{attribute 'qualified_only'}
VAR_GLOBAL
	OutputData AT %Q*: ARRAY[0..7] OF BYTE;
	
	InputData1 AT %I*: ARRAY[0..7] OF BYTE;
	InputData2 AT %I*: ARRAY[0..7] OF BYTE;
	InputData3 AT %I*: ARRAY[0..7] OF BYTE;
	state AT %I* : UINT;
	
	EHWTable1XML : STRING[6000];

	TrackSegmentsRaw1 : ARRAY[0..29] OF ST_Track_Segment_Raw_EHC:= [
		(iTrackNumber := 1, iXPosition := 0, sType := "straight", sBatch := "B", iId := 61, iLength := 4, rStartValue := 640.0, rEndValue := 644.0),
(iTrackNumber := 2, iXPosition := 4, sType := "straight", sBatch := "B", iId := 58, iLength := 4, rStartValue := 628.0, rEndValue := 632.0),
(iTrackNumber := 3, iXPosition := 8, sType := "straight", sBatch := "B", iId := 60, iLength := 4, rStartValue := 636.0, rEndValue := 640.0),
(iTrackNumber := 4, iXPosition := 12, sType := "straight", sBatch := "B", iId := 24, iLength := 4.2, rStartValue := 304.6, rEndValue := 308.8),
(iTrackNumber := 5, iXPosition := 16.4, sType := "straight", sBatch := "B", iId := 2, iLength := 4.2, rStartValue := 212.2, rEndValue := 216.4),
(iTrackNumber := 6, iXPosition := 20.6, sType := "straight", sBatch := "B", iId := 66, iLength := 4, rStartValue := 660.0, rEndValue := 664.0),
(iTrackNumber := 7, iXPosition := 24.6, sType := "straight", sBatch := "B", iId := 65, iLength := 4, rStartValue := 656.0, rEndValue := 660.0),
(iTrackNumber := 8, iXPosition := 28.6, sType := "straight", sBatch := "B", iId := 55, iLength := 4, rStartValue := 616.0, rEndValue := 620.0),
(iTrackNumber := 9, iXPosition := 32.6, sType := "straight", sBatch := "B", iId := 47, iLength := 4, rStartValue := 584.0, rEndValue := 588.0),
(iTrackNumber := 10, iXPosition := 36.6, sType := "straight", sBatch := "B", iId := 44, iLength := 4, rStartValue := 572.0, rEndValue := 576.0),
(iTrackNumber := 11, iXPosition := 40.6, sType := "straight", sBatch := "B", iId := 178, iLength := 4, rStartValue := 1108.0, rEndValue := 1112.0),
(iTrackNumber := 12, iXPosition := 44.6, sType := "straight", sBatch := "B", iId := 4, iLength := 4.2, rStartValue := 220.6, rEndValue := 224.8),
(iTrackNumber := 13, iXPosition := 49, sType := "straight", sBatch := "B", iId := 9, iLength := 4.2, rStartValue := 241.6, rEndValue := 245.8),
(iTrackNumber := 14, iXPosition := 53.2, sType := "straight", sBatch := "B", iId := 181, iLength := 4, rStartValue := 1120.0, rEndValue := 1124.0),
(iTrackNumber := 15, iXPosition := 57.2, sType := "straight", sBatch := "B", iId := 164, iLength := 4, rStartValue := 1052.0, rEndValue := 1056.0),
(iTrackNumber := 16, iXPosition := 61.2, sType := "straight", sBatch := "B", iId := 74, iLength := 4, rStartValue := 692.0, rEndValue := 696.0),
(iTrackNumber := 17, iXPosition := 65.2, sType := "straight", sBatch := "B", iId := 166, iLength := 4, rStartValue := 1060.0, rEndValue := 1064.0),
(iTrackNumber := 18, iXPosition := 69.2, sType := "straight", sBatch := "B", iId := 32, iLength := 4, rStartValue := 524.0, rEndValue := 528.0),
(iTrackNumber := 19, iXPosition := 73.2, sType := "straight", sBatch := "B", iId := 184, iLength := 4, rStartValue := 1132.0, rEndValue := 1136.0),
(iTrackNumber := 20, iXPosition := 77.2, sType := "straight", sBatch := "B", iId := 187, iLength := 4, rStartValue := 1144.0, rEndValue := 1148.0),
(iTrackNumber := 21, iXPosition := 81.2, sType := "straight", sBatch := "B", iId := 16, iLength := 4, rStartValue := 460.0, rEndValue := 464.0),
(iTrackNumber := 22, iXPosition := 85.2, sType := "straight", sBatch := "B", iId := 14, iLength := 4, rStartValue := 452.0, rEndValue := 456.0),
(iTrackNumber := 23, iXPosition := 89.2, sType := "straight", sBatch := "B", iId := 13, iLength := 4, rStartValue := 448.0, rEndValue := 452.0),
(iTrackNumber := 24, iXPosition := 93.2, sType := "straight", sBatch := "B", iId := 22, iLength := 4, rStartValue := 484.0, rEndValue := 488.0),
(iTrackNumber := 25, iXPosition := 97.2, sType := "straight", sBatch := "B", iId := 158, iLength := 4, rStartValue := 1028.0, rEndValue := 1032.0),
(iTrackNumber := 26, iXPosition := 101.2, sType := "straight", sBatch := "B", iId := 38, iLength := 4, rStartValue := 548.0, rEndValue := 552.0),
(iTrackNumber := 27, iXPosition := 105.2, sType := "straight", sBatch := "B", iId := 120, iLength := 4, rStartValue := 876.0, rEndValue := 880.0),
(iTrackNumber := 28, iXPosition := 109.2, sType := "straight", sBatch := "B", iId := 20, iLength := 4.2, rStartValue := 287.8, rEndValue := 292.0)
	];
END_VAR

(* stored: Version 1.1.0.1
   GVL GVL_PROP_BARCODE: Id {dacfeddd-689b-44e3-a4fb-78e29b4ae552} *)
